// ==============================================================================
// FB_Test_Valve3P - РўРµСЃС‚РѕРІРёР№ Р±Р»РѕРє РґР»СЏ Valve3P (С‚СЂРёРїРѕР·РёС†С–Р№РЅРёР№ РєР»Р°РїР°РЅ)
// ==============================================================================
// Р’РµСЂСЃС–СЏ: 1.0.0
// Р”Р°С‚Р°: 2026-03-27
// ==============================================================================
// РџСЂРёР·РЅР°С‡РµРЅРЅСЏ:
//   Unit-С‚РµСЃС‚Рё РґР»СЏ FC_Valve3P Р·Р° Р°РЅР°Р»РѕРіС–С”СЋ Р· FB_Test_Gate2P
//
// Р’РёРєРѕСЂРёСЃС‚Р°РЅРЅСЏ:
//   "FB_Test_Valve3P"(
//       Run    := TRUE,      // РІРёРєРѕРЅР°С‚Рё С‚РµСЃС‚
//       CaseId := 1          // РЅРѕРјРµСЂ С‚РµСЃС‚-РєРµР№СЃСѓ
//   );
//   // РџРµСЂРµРІС–СЂРёС‚Рё: Passed, Failed, FailMask
// ==============================================================================
FUNCTION_BLOCK "FB_Test_Valve3P"
{ S7_Optimized_Access := 'TRUE' }
VERSION : 1.0

VAR_INPUT
    Run : Bool;   // TRUE = РІРёРєРѕРЅР°С‚Рё С‚РµСЃС‚
    CaseId : Int;   // РЅРѕРјРµСЂ С‚РµСЃС‚-РєРµР№СЃСѓ
END_VAR

VAR_OUTPUT
    Passed : Bool;
    Failed : Bool;
    FailMask : DWord;
END_VAR

VAR
    F : "UDT_Valve3P";
    B : "UDT_BaseMechanism";
    now : DInt;   // РїРѕС‚РѕС‡РЅРёР№ С‡Р°СЃ (TIME_TCK)

    // РћС‡С–РєСѓРІР°РЅРЅСЏ
    Exp_Status : UInt;
    Exp_FLTCode : UInt;
    Exp_DO_Pos0 : Bool;
    Exp_DO_Pos1 : Bool;
    Exp_DO_Pos2 : Bool;
END_VAR


BEGIN

    #Passed := FALSE;
    #Failed := FALSE;
    #FailMask := 0;

    IF NOT #Run THEN
        RETURN;
    END_IF;

    #now := TIME_TCK();

    // ==============================================================================
    // ARRANGE вЂ” Р±Р°Р·РѕРІРёР№ "Р·РґРѕСЂРѕРІРёР№" СЃС‚Р°РЅ
    // ==============================================================================

    // Base
    #B.Enable_OK := TRUE;
    #B.LocalManual := FALSE;
    #B.DeviceType := "TYPE_VALVE3P";
    #B.Cmd := "CMD_NONE";
    #B.CmdParam1 := 0;
    #B.LastCmd := "CMD_NONE";
    #B.Force_Code := 0;
    #B.OwnerCur := 123;  // РїРµСЂРµРІС–СЂРёРјРѕ С‰Рѕ РєРёРґР°С”
    #B.OwnerCurId := 456;
    #B.Status := "STS_IDLE";
    #B.FLTCode := "FLT_NONE";

    // РўР°Р№РјС–РЅРіРё
    #F.MoveStartMs := 0;
    #F.UnknownPositionMs := 0;

    // HAL
    #F.DI_Breaker_OK := TRUE;
    #F.DI_Pos0_OK := FALSE;
    #F.DI_Pos1_OK := FALSE;
    #F.DI_Pos2_OK := FALSE;

    // Р”РµС„РѕР»С‚ РѕС‡С–РєСѓРІР°РЅСЊ
    #Exp_Status := #B.Status;
    #Exp_FLTCode := #B.FLTCode;
    #Exp_DO_Pos0 := FALSE;
    #Exp_DO_Pos1 := FALSE;
    #Exp_DO_Pos2 := FALSE;

    // ==============================================================================
    // TEST CASES
    // ==============================================================================
    CASE #CaseId OF

        // ======================================================================
        // A1: Enable_OK = FALSE в†’ DISABLED
        // ======================================================================
        1:
            #B.Enable_OK := FALSE;
            #Exp_Status := "STS_DISABLED";

        // ======================================================================
        // A2: LocalManual = TRUE в†’ LOCAL
        // ======================================================================
        2:
            #B.LocalManual := TRUE;
            #Exp_Status := "STS_LOCAL";

        // ======================================================================
        // B1: RESET СЃРєРёРґР°С” FAULT С– С‚Р°Р№РјС–РЅРіРё
        // ======================================================================
        3:
            #B.Status := "STS_FAULT";
            #B.FLTCode := "FLT_VALVE_MOVE_TIMEOUT";
            #F.MoveStartMs := 111;
            #F.UnknownPositionMs := 2323;
            #B.Cmd := "CMD_RESET";
            #Exp_Status := "STS_IDLE";
            #Exp_FLTCode := "FLT_NONE";
            // РџСЂРёРјС–С‚РєР°: UnknownPositionMs СЃРєРёРґР°С”С‚СЊСЃСЏ С‚С–Р»СЊРєРё СЏРєС‰Рѕ Р±СѓР»Р° Unknown РїРѕР·РёС†С–СЏ
            // РЈ С†СЊРѕРјСѓ С‚РµСЃС‚С– FLT_VALVE_MOVE_TIMEOUT СЃРєРёРґР°С”С‚СЊСЃСЏ Р·Р°РІР¶РґРё (РЅРµРјР°С” С„С–Р·. РґР°С‚С‡РёРєР°)

        // ======================================================================
        // C1: Breaker Р°РІР°СЂС–СЏ
        // ======================================================================
        4:
            #F.DI_Breaker_OK := FALSE;
            #Exp_Status := "STS_FAULT";
            #Exp_FLTCode := "FLT_BREAKER";

        // ======================================================================
        // C2: Unknown Position (РЅРµРІС–РґРѕРјР° РїРѕР·РёС†С–СЏ > С‚Р°Р№РјР°СѓС‚)
        // ======================================================================
        5:
            #B.Status := "STS_IDLE";
            #F.DI_Pos0_OK := FALSE;
            #F.DI_Pos1_OK := FALSE;
            #F.DI_Pos2_OK := FALSE;
            #F.UnknownPositionMs := #now - "TimeoutMs_Valve_Position_Unknown" - 1;
            #Exp_Status := "STS_FAULT";
            #Exp_FLTCode := "FLT_VALVE_POS_UNKNOWN";

        // ======================================================================
        // C3: Breaker > Unknown Position (РїСЂС–РѕСЂРёС‚РµС‚ Breaker)
        // ======================================================================
        6:
            #B.Status := "STS_IDLE";
            #F.DI_Breaker_OK := FALSE;
            #F.DI_Pos0_OK := FALSE;
            #F.DI_Pos1_OK := FALSE;
            #F.DI_Pos2_OK := FALSE;
            #F.UnknownPositionMs := #now - "TimeoutMs_Valve_Position_Unknown" - 1;
            #Exp_Status := "STS_FAULT";
            #Exp_FLTCode := "FLT_BREAKER";

        // ======================================================================
        // C4: Multiple Positions (2+ РґР°С‚С‡РёРєС–РІ Р°РєС‚РёРІРЅС–)
        // ======================================================================
        7:
            #F.DI_Pos0_OK := TRUE;
            #F.DI_Pos1_OK := TRUE;
            #F.DI_Pos2_OK := FALSE;
            #Exp_Status := "STS_FAULT";
            #Exp_FLTCode := "FLT_VALVE_MULTIPLE_POS";

        // ======================================================================
        // C5: Multiple Positions (РІСЃС– 3 Р°РєС‚РёРІРЅС–)
        // ======================================================================
        8:
            #F.DI_Pos0_OK := TRUE;
            #F.DI_Pos1_OK := TRUE;
            #F.DI_Pos2_OK := TRUE;
            #Exp_Status := "STS_FAULT";
            #Exp_FLTCode := "FLT_VALVE_MULTIPLE_POS";

        // ======================================================================
        // D1: Р¤РѕСЂСЃСѓРІР°РЅРЅСЏ BREAKER
        // ======================================================================
        9:
            #F.DI_Breaker_OK := FALSE;
            #B.Force_Code := 1;  // BIT0 = forceBreaker
            #Exp_Status := "STS_IDLE";
            #Exp_FLTCode := "FLT_NONE";  // Р¤РѕСЂСЃСѓРІР°РЅРЅСЏ СЃРєРёРґР°С” FLTCode
            #Exp_DO_Pos0 := FALSE;
            #Exp_DO_Pos1 := FALSE;
            #Exp_DO_Pos2 := FALSE;

        // ======================================================================
        // D2: Р¤РѕСЂСЃСѓРІР°РЅРЅСЏ VALVE_POS_UNKNOWN
        // ======================================================================
        10:
            #B.Force_Code := 32;  // BIT5 = forcePosUnknown
            #B.Status := "STS_IDLE";
            #B.FLTCode := "FLT_NONE";  // РЇРІРЅРѕ СЃРєРёРґР°С”РјРѕ FLTCode РЅР° РїРѕС‡Р°С‚РєСѓ
            #F.DI_Pos0_OK := FALSE;
            #F.DI_Pos1_OK := FALSE;
            #F.DI_Pos2_OK := FALSE;
            #F.UnknownPositionMs := #now - "TimeoutMs_Valve_Position_Unknown" - 1;
            #Exp_Status := "STS_IDLE";
            #Exp_FLTCode := "FLT_NONE";  // Р¤РѕСЂСЃСѓРІР°РЅРЅСЏ СЃРєРёРґР°С” FLTCode
            #Exp_DO_Pos0 := FALSE;
            #Exp_DO_Pos1 := FALSE;
            #Exp_DO_Pos2 := FALSE;

        // ======================================================================
        // D3: Р¤РѕСЂСЃСѓРІР°РЅРЅСЏ VALVE_MOVE_TIMEOUT
        // ======================================================================
        11:
            #B.Force_Code := 16;  // BIT4 = forceMoveTimeout
            #B.Status := "STS_RUNNING";
            #B.FLTCode := "FLT_NONE";  // РЇРІРЅРѕ СЃРєРёРґР°С”РјРѕ FLTCode РЅР° РїРѕС‡Р°С‚РєСѓ
            #B.CmdParam1 := "CMD_VALVE_POS1";
            #F.DO_Pos1 := TRUE;  // Р’СЃС‚Р°РЅРѕРІР»СЋС”РјРѕ РїРµСЂРµРґ С‚РµСЃС‚РѕРј
            #F.MoveStartMs := #now - "TimeoutMs_Valve_Move" - 1;
            #Exp_Status := "STS_RUNNING";
            #Exp_FLTCode := "FLT_NONE";  // Р¤РѕСЂСЃСѓРІР°РЅРЅСЏ СЃРєРёРґР°С” FLTCode
            #Exp_DO_Pos0 := FALSE;
            #Exp_DO_Pos1 := TRUE;  // Р’РёС…С–Рґ Р·Р°Р»РёС€Р°С”С‚СЊСЃСЏ Р°РєС‚РёРІРЅРёРј
            #Exp_DO_Pos2 := FALSE;

        // ======================================================================
        // E1: START + CMD_VALVE_POS0 + DI_Pos0_OK в†’ IDLE (РІР¶Рµ Сѓ РїРѕР·РёС†С–С—)
        // ======================================================================
        12:
            #B.Cmd := "CMD_START";
            #B.CmdParam1 := "CMD_VALVE_POS0";
            #F.DI_Pos0_OK := TRUE;
            #Exp_Status := "STS_IDLE";
            #Exp_DO_Pos0 := FALSE;
            #Exp_DO_Pos1 := FALSE;
            #Exp_DO_Pos2 := FALSE;

        // ======================================================================
        // E2: START + CMD_VALVE_POS1 + DI_Pos1_OK в†’ IDLE (РІР¶Рµ Сѓ РїРѕР·РёС†С–С—)
        // ======================================================================
        13:
            #B.Cmd := "CMD_START";
            #B.CmdParam1 := "CMD_VALVE_POS1";
            #F.DI_Pos1_OK := TRUE;
            #Exp_Status := "STS_IDLE";
            #Exp_DO_Pos0 := FALSE;
            #Exp_DO_Pos1 := FALSE;
            #Exp_DO_Pos2 := FALSE;

        // ======================================================================
        // E3: START + CMD_VALVE_POS2 + DI_Pos2_OK в†’ IDLE (РІР¶Рµ Сѓ РїРѕР·РёС†С–С—)
        // ======================================================================
        14:
            #B.Cmd := "CMD_START";
            #B.CmdParam1 := "CMD_VALVE_POS2";
            #F.DI_Pos2_OK := TRUE;
            #Exp_Status := "STS_IDLE";
            #Exp_DO_Pos0 := FALSE;
            #Exp_DO_Pos1 := FALSE;
            #Exp_DO_Pos2 := FALSE;

        // ======================================================================
        // E4: START + CMD_VALVE_POS0 + Not DI_Pos0_OK в†’ STARTING
        // ======================================================================
        15:
            #B.Cmd := "CMD_START";
            #B.CmdParam1 := "CMD_VALVE_POS0";
            #F.DI_Pos0_OK := FALSE;
            #Exp_Status := "STS_STARTING";
            #Exp_DO_Pos0 := TRUE;
            #Exp_DO_Pos1 := FALSE;
            #Exp_DO_Pos2 := FALSE;

        // ======================================================================
        // E5: START + CMD_VALVE_POS1 + Not DI_Pos1_OK в†’ STARTING
        // ======================================================================
        16:
            #B.Cmd := "CMD_START";
            #B.CmdParam1 := "CMD_VALVE_POS1";
            #F.DI_Pos1_OK := FALSE;
            #Exp_Status := "STS_STARTING";
            #Exp_DO_Pos0 := FALSE;
            #Exp_DO_Pos1 := TRUE;
            #Exp_DO_Pos2 := FALSE;

        // ======================================================================
        // E6: START + CMD_VALVE_POS2 + Not DI_Pos2_OK в†’ STARTING
        // ======================================================================
        17:
            #B.Cmd := "CMD_START";
            #B.CmdParam1 := "CMD_VALVE_POS2";
            #F.DI_Pos2_OK := FALSE;
            #Exp_Status := "STS_STARTING";
            #Exp_DO_Pos0 := FALSE;
            #Exp_DO_Pos1 := FALSE;
            #Exp_DO_Pos2 := TRUE;

        // ======================================================================
        // E7: STARTING + Not DI_Pos0_OK в†’ RUNNING (Р·С–Р№С€РѕРІ Р· РєС–РЅС†РµРІРёРєР°)
        // ======================================================================
        18:
            #B.Status := "STS_STARTING";
            #B.CmdParam1 := "CMD_VALVE_POS0";
            #F.DI_Pos0_OK := FALSE;
            #Exp_Status := "STS_RUNNING";
            #Exp_DO_Pos0 := TRUE;
            #Exp_DO_Pos1 := FALSE;
            #Exp_DO_Pos2 := FALSE;

        // ======================================================================
        // E8: STARTING + DI_Pos0_OK в†’ IDLE (РЅРµ Р·С–Р№С€Р»Р°, РІР¶Рµ Сѓ РїРѕР·РёС†С–С—)
        // ======================================================================
        19:
            #B.Status := "STS_STARTING";
            #B.CmdParam1 := "CMD_VALVE_POS0";
            #F.DI_Pos0_OK := TRUE;
            #Exp_Status := "STS_IDLE";
            #Exp_DO_Pos0 := FALSE;
            #Exp_DO_Pos1 := FALSE;
            #Exp_DO_Pos2 := FALSE;

        // ======================================================================
        // E9: RUNNING + MoveTimeout в†’ FLT_VALVE_MOVE_TIMEOUT
        // ======================================================================
        20:
            #B.Status := "STS_RUNNING";
            #B.CmdParam1 := "CMD_VALVE_POS1";
            #F.DO_Pos1 := TRUE;
            #F.MoveStartMs := #now - "TimeoutMs_Valve_Move" - 1;
            #Exp_Status := "STS_FAULT";
            #Exp_FLTCode := "FLT_VALVE_MOVE_TIMEOUT";
            #Exp_DO_Pos0 := FALSE;
            #Exp_DO_Pos1 := FALSE;
            #Exp_DO_Pos2 := FALSE;

        // ======================================================================
        // E10: RUNNING + РґРѕСЃСЏРіРЅСѓС‚Рѕ РїРѕР·РёС†С–С— в†’ STOPPING
        // ======================================================================
        21:
            #B.Status := "STS_RUNNING";
            #B.FLTCode := "FLT_NONE";  // РЇРІРЅРѕ СЃРєРёРґР°С”РјРѕ FLTCode
            #B.CmdParam1 := "CMD_VALVE_POS1";
            #F.DI_Pos1_OK := TRUE;
            #F.MoveStartMs := 0;  // РЎРєРёРґР°С”РјРѕ С‚Р°Р№РјРµСЂ СЂСѓС…Сѓ (С‰Рµ РЅРµ С‡Р°СЃ С‚Р°Р№РјР°СѓС‚Сѓ)
            #Exp_Status := "STS_STOPPING";
            #Exp_FLTCode := "FLT_NONE";
            #Exp_DO_Pos0 := FALSE;
            #Exp_DO_Pos1 := FALSE;
            #Exp_DO_Pos2 := FALSE;

        // ======================================================================
        // E11: STOPPING + DI_Pos1_OK в†’ IDLE
        // ======================================================================
        22:
            #B.Status := "STS_STOPPING";
            #F.DI_Pos1_OK := TRUE;
            #Exp_Status := "STS_IDLE";
            #Exp_DO_Pos0 := FALSE;
            #Exp_DO_Pos1 := FALSE;
            #Exp_DO_Pos2 := FALSE;

        // ======================================================================
        // E12: STOP РїС–Рґ С‡Р°СЃ STARTING в†’ STOPPING
        // ======================================================================
        23:
            #B.Status := "STS_STARTING";
            #B.Cmd := "CMD_STOP";
            #Exp_Status := "STS_STOPPING";

        // ======================================================================
        // E13: STOP РїС–Рґ С‡Р°СЃ RUNNING в†’ STOPPING
        // ======================================================================
        24:
            #B.Status := "STS_RUNNING";
            #B.FLTCode := "FLT_NONE";  // РЇРІРЅРѕ СЃРєРёРґР°С”РјРѕ FLTCode
            #B.Cmd := "CMD_STOP";
            #F.DI_Pos0_OK := FALSE;  // РљР»Р°РїР°РЅ Сѓ СЂСѓСЃС– (РЅРµРјР°С” РїРѕР·РёС†С–С—)
            #F.DI_Pos1_OK := FALSE;
            #F.DI_Pos2_OK := FALSE;
            #F.MoveStartMs := 0;  // РЎРєРёРґР°С”РјРѕ С‚Р°Р№РјРµСЂ СЂСѓС…Сѓ (С‰Рµ РЅРµ С‡Р°СЃ С‚Р°Р№РјР°СѓС‚Сѓ)
            #Exp_Status := "STS_STOPPING";
            #Exp_FLTCode := "FLT_NONE";

        // ======================================================================
        // E14: Р’С–РґРЅРѕРІР»РµРЅРЅСЏ Р· DISABLED в†’ IDLE
        // ======================================================================
        25:
            #B.Status := "STS_DISABLED";
            #B.Enable_OK := TRUE;
            #Exp_Status := "STS_IDLE";

        // ======================================================================
        // E15: Р’С–РґРЅРѕРІР»РµРЅРЅСЏ Р· LOCAL в†’ IDLE
        // ======================================================================
        26:
            #B.Status := "STS_LOCAL";
            #B.LocalManual := FALSE;
            #Exp_Status := "STS_IDLE";

        ELSE
            RETURN;
    END_CASE;

    // ==============================================================================
    // ACT вЂ” РІРёРєР»РёРє С„СѓРЅРєС†С–С— РєРµСЂСѓРІР°РЅРЅСЏ
    // ==============================================================================
    "FC_Valve3P"(
        F := #F,
        B := #B
    );

    // ==============================================================================
    // ASSERT вЂ” РїРµСЂРµРІС–СЂРєР° СЂРµР·СѓР»СЊС‚Р°С‚С–РІ
    // ==============================================================================
    IF #B.Status <> #Exp_Status THEN
        #FailMask := #FailMask OR 16#0001;
    END_IF;

    IF #B.FLTCode <> #Exp_FLTCode THEN
        #FailMask := #FailMask OR 16#0002;
    END_IF;

    IF #F.DO_Pos0 <> #Exp_DO_Pos0 THEN
        #FailMask := #FailMask OR 16#0004;
    END_IF;

    IF #F.DO_Pos1 <> #Exp_DO_Pos1 THEN
        #FailMask := #FailMask OR 16#0008;
    END_IF;

    IF #F.DO_Pos2 <> #Exp_DO_Pos2 THEN
        #FailMask := #FailMask OR 16#0010;
    END_IF;

    // RESET РґРѕРґР°С‚РєРѕРІС– РіР°СЂР°РЅС‚С–С— (С‚Р°Р№РјС–РЅРіРё РїРѕРІРёРЅРЅС– РѕР±РЅСѓР»РёС‚РёСЃСЏ)
    IF #CaseId = 3 THEN
        IF #F.MoveStartMs <> 0 THEN
            #FailMask := #FailMask OR 16#0020;
        END_IF;
        // UnknownPositionMs СЃРєРёРґР°С”С‚СЊСЃСЏ С‚С–Р»СЊРєРё СЏРєС‰Рѕ FLTCode Р±СѓРІ FLT_VALVE_POS_UNKNOWN
        // РЈ С†СЊРѕРјСѓ С‚РµСЃС‚С– FLT_VALVE_MOVE_TIMEOUT в†’ UnknownPositionMs РЅРµ С‡С–РїР°С”С‚СЊСЃСЏ
        // РўРѕРјСѓ РїРµСЂРµРІС–СЂСЏС”РјРѕ С‚С–Р»СЊРєРё MoveStartMs
    END_IF;

    #Failed := (#FailMask <> 0);
    #Passed := NOT #Failed;

END_FUNCTION_BLOCK
